# EPICS substitutions: ek9000App/Db/EL2124.substitutions
file EL2124.template
{       pattern
        {
                TERMINAL,

        }
        {
        }
}
